// Mitsubishi GX Works2 project: k05   PLC: Q02/Q02H

PROGRAM MAIN
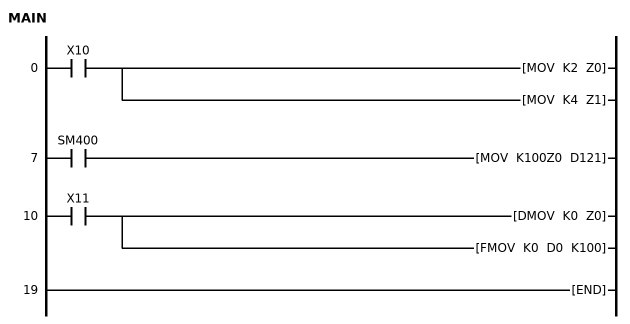
0     LD      X10
      MOV     K2 Z0
      MOV     K4 Z1
7     LD      SM400
      MOV     K100Z0 D121
10    LD      X11
      DMOV    K0 Z0
      FMOV    K0 D0 K100
19    END
END_PROGRAM
